(* IEC 61131-3 sources: AXOpen/src/components.rexroth.drives/ctrl/src/AxoIndraDrive (part 2) *)

            _AxisReference ?= AxisRef;

            Messenger.ActivateOnCondition(ULINT#1401,_AxisReference = NULL, eAxoMessageCategory#ProgrammingError);

            IF(_AxisReference = NULL) THEN
                RETURN;
            END_IF;

            Status := FALSE;
            Error	:= FALSE;
            ErrorID :=	DINT#0;
            Valid := FALSE;
            IF Enable OR MC_PowerEnable_PV THEN
                IF _AxisReference^.Data.CheckAccessOK	THEN
                    IF Enable THEN (*	raising edge of ENABLE *)
                        _AxisReference^.Data.PowerOnReq := TRUE;
                    ELSE
                        _AxisReference^.Data.PowerOnReq := FALSE;
                        _AxisReference^.Data.CallNumberCyclic := _AxisReference^.Data.CallNumberCyclic + INT#2;
                    END_IF;
                    _AxisReference^.Data.CallAxis := TRUE;
                    _AxisReference^.Data.ReadOnlyData := FALSE;
                        THIS.FieldBusCommunication(AxisRef := _AxisReference,
                                                    CommandWriteActive=> Dummy);
                    IF _AxisReference^.Data.PowerOK THEN
                        Status	:= TRUE;						(* Status OK*)
                        Valid := TRUE;
                    END_IF;
                    IF _AxisReference^.Data.PowerError = TRUE THEN
                        Error		:= TRUE; 						(*	Set the ERROR-Output *)
                        Valid := TRUE;
                        ErrorID := TO_DINT(_AxisReference^.Data.ErrorID);
                    ELSIF _AxisReference^.Data.CallAxis THEN
                        Error := TRUE;
                        Valid := TRUE;
                        ErrorID := TO_DINT(AXOpen.Components.Rexroth.Drives.eAxoIndraDriveErrorCode#RESOURCE_ERROR);
                    END_IF;
                ELSE
                    Error := TRUE;
                    Valid := TRUE;
                    ErrorID :=TO_DINT( AXOpen.Components.Rexroth.Drives.eAxoIndraDriveErrorCode#RESOURCE_ERROR);
                END_IF;
            END_IF;
            MC_PowerEnable_PV := Enable;
        END_METHOD

        ///<summary>
        /// This method commands the axis to perform the «search home» sequence. The details of this sequence are
        /// manufacturer dependent and can be set by the axis’ parameters. The ‘Position’ input is used to set the absolute
        /// position when reference signal is detected. This method completes at ‘Standstill’ if it was started in ‘Standstill’.
        ///</summary>
        VAR INTERNAL
            MC_HomeExecute_PV					:	BOOL := FALSE;		//Execute - previous value
            MC_HomeCallNumber					: 	INT; 				//Call number of the method MC_Stop
            MC_HomeFirstCall					: 	BOOL;				//First call of the method MC_Stop
            MC_HomeDone_						:	BOOL;
            MC_HomeActive_						:	BOOL;
            MC_HomeCommandAborted_				:	BOOL;
            MC_HomeError_						:	BOOL;
            MC_HomeErrorID_						:	DINT;
            MC_HomeState_						:	UINT;
        END_VAR
        METHOD PUBLIC OVERRIDE MC_Home
            VAR_INPUT
                AxisRef         :   AXOpen.Components.Abstractions.Drives.IAxoAxisReference;
                Execute         :   BOOL;                       //  Start the motion at rising edge
                Position        :   LREAL;                      //  Absolute position when the reference signal is detected
                HommingMode     :   INT;                        //  Required homming mode
                Velocity        :   LREAL;                      //  Value of the maximum ‘Velocity’ (not necessarily reached) [u/s].
                Acceleration    :   LREAL;                      //  Value of the ‘Acceleration’ (always positive) (increasing energy of the motor) [u/s2]
                Deceleration    :   LREAL;                      //  Value of the ‘Deceleration’ (always positive) (decreasing energy of the motor) [u/s2]
            END_VAR
            VAR_OUTPUT
                Done            :   BOOL;                       // Reference known and set sucessfully
                Busy            :   BOOL;                       // The method is not finished and new output values are to be expected
                Active          :   BOOL;                       // Indicates that the method has control on the axis
                CommandAborted  :   BOOL;                       // ‘Command’ is aborted by another command
                Error           :   BOOL;                       // Signals that an error has occurred within the method
                ErrorID         :   DINT;                       // Error identification
             END_VAR
             VAR
                _AxisReference :  REF_TO AXOpen.Components.Rexroth.Drives.AxoIndraDriveAxisReference;

                _ErrorID : DINT;
                _HommingMode: DINT;
                Dummy : BOOL;
                _result : IAxoTaskState;
            END_VAR

            _AxisReference ?= AxisRef;

            Messenger.ActivateOnCondition(ULINT#1402,_AxisReference = NULL, eAxoMessageCategory#ProgrammingError);

            IF(_AxisReference = NULL) THEN
                RETURN;
            END_IF;

            IF Execute AND NOT MC_HomeExecute_PV AND MC_HomeState_ = UINT#0 THEN
                MC_HomeState_ := UINT#10;
            END_IF;
            IF MC_HomeState_ = UINT#10 THEN
                //S-0-0052, Reference distance of encoder 1
                _result := THIS.AxoWriteParameter(ParameterNumber := 52, Value := TO_DINT(Position * EXP(LN(10)* PositionExponent)),ExecutionMode := AXOpen.Components.Abstractions.Drives.eAxoExecutionMode#Immediately, ErrorID =>_ErrorID);
                IF _result.IsDone() THEN
                    MC_HomeState_ := UINT#20;
                END_IF;
                IF _result.HasError() THEN
                    MC_HomeError_ := TRUE;
                    MC_HomeErrorID_ := _ErrorID;
                END_IF;
            END_IF;
            IF MC_HomeState_ = UINT#20 THEN
                AxoWriteParameter_Task.Restore();
                IF(AxoWriteParameter_Task.IsReady()) THEN
                    MC_HomeState_ :=UINT#30;
                    RETURN;
                END_IF;
            END_IF;
            IF MC_HomeState_ = UINT#30 THEN
                IF HommingMode = 0 THEN
                    _HommingMode := 551;
                ELSE
                    _HommingMode := HommingMode;
                END_IF;
                //S-0-0147, Homing parameter
                _result := THIS.AxoWriteParameter(ParameterNumber := 147, Value := _HommingMode ,ExecutionMode := AXOpen.Components.Abstractions.Drives.eAxoExecutionMode#Immediately,ErrorID =>_ErrorID);
                IF _result.IsDone() THEN
                    MC_HomeState_ := UINT#40;
                END_IF;
                IF _result.HasError() THEN
                    MC_HomeError_ := TRUE;
                    MC_HomeErrorID_ := _ErrorID;
                END_IF;
            END_IF;
            IF MC_HomeState_ = UINT#40 THEN
                AxoWriteParameter_Task.Restore();
                IF(AxoWriteParameter_Task.IsReady()) THEN
                    MC_HomeState_ := UINT#50;
                    RETURN;
                END_IF;
            END_IF;
            IF MC_HomeState_ = UINT#50 THEN
                //S-0-0041, Homing velocity
                _result := THIS.AxoWriteParameter(ParameterNumber := 41, Value := TO_DINT(Velocity * EXP(LN(10)*VelocityExponent)) ,ExecutionMode := AXOpen.Components.Abstractions.Drives.eAxoExecutionMode#Immediately, ErrorID =>_ErrorID);
                IF _result.IsDone() THEN
                    MC_HomeState_ :=UINT#60;
                END_IF;
                IF _result.HasError() THEN
                    MC_HomeError_ := TRUE;
                    MC_HomeErrorID_ := _ErrorID;
                END_IF;
            END_IF;
            IF MC_HomeState_ = UINT#60 THEN
                AxoWriteParameter_Task.Restore();
                IF(AxoWriteParameter_Task.IsReady()) THEN
                    MC_HomeState_ :=UINT#70;
                    RETURN;
                END_IF;
            END_IF;
            IF MC_HomeState_ = UINT#70 THEN
                //S-0-0042, Homing acceleration
                _result := THIS.AxoWriteParameter(ParameterNumber := 42, Value := TO_DINT(Acceleration * EXP(LN(10)*AccelerationExponent)) ,ExecutionMode := AXOpen.Components.Abstractions.Drives.eAxoExecutionMode#Immediately, ErrorID =>_ErrorID);
                IF _result.IsDone() THEN
                    MC_HomeState_ := UINT#80;
                END_IF;
                IF _result.HasError() THEN
                    MC_HomeError_ := TRUE;
                    MC_HomeErrorID_ := _ErrorID;
                END_IF;
            END_IF;
            IF MC_HomeState_ = UINT#80 THEN
                AxoWriteParameter_Task.Restore();
                IF(AxoWriteParameter_Task.IsReady()) THEN
                    MC_HomeState_ := UINT#90;
                    RETURN;
                END_IF;
            END_IF;

            IF Execute AND MC_HomeState_ < UINT#90 THEN
                RETURN;
            END_IF;

            (************ start of homing *****************************)
            IF Execute OR MC_HomeExecute_PV  THEN
                MC_HomeFirstCall := TRUE;
                IF _AxisReference^.Data.CheckAccessOK	THEN
                    IF NOT _AxisReference^.Data.PowerOK OR  _AxisReference^.Data.DriveStopReq AND MC_HomeActive_ THEN
                        MC_HomeDone_ := FALSE;
                        MC_HomeActive_ := FALSE;
                        MC_HomeCommandAborted_ := TRUE;
                        _AxisReference^.Data.HomingReq:= FALSE;
                    END_IF;
                    IF Execute AND NOT MC_HomeExecute_PV  THEN
                        IF _AxisReference^.Data.PowerOK AND NOT _AxisReference^.Data.DriveStopReq THEN
                            _AxisReference^.Data.CallNumberCyclic := _AxisReference^.Data.CallNumberCyclic + INT#2;
                            MC_HomeCallNumber := _AxisReference^.Data.CallNumberCyclic;
                            _AxisReference^.Data.WriteCommand:= TRUE;
                            _AxisReference^.Data.HomingReq:= TRUE;
                            _AxisReference^.Data.DriveStopReq:= FALSE;
                            _AxisReference^.Data.DriveHaltReq:= FALSE;
                            _AxisReference^.Data.MoveVelocityReq:= FALSE;
                            _AxisReference^.Data.TorqueControlReq:= FALSE;
                            _AxisReference^.Data.Relative:= FALSE;
                            _AxisReference^.Data.Additive:= FALSE;
                            _AxisReference^.Data.Position := Position;
                            _AxisReference^.Data.Velocity := Velocity;
                            _AxisReference^.Data.Acceleration := Acceleration;
                            _AxisReference^.Data.Deceleration := Deceleration;
                        ELSE
                            MC_HomeError_ := TRUE;
                            MC_HomeErrorID_ := TO_DINT(AXOpen.Components.Rexroth.Drives.eAxoIndraDriveErrorCode#STATE_MACHINE_Error); 	(*State machine MC_HomeError_*)
                        END_IF;
                    END_IF;
                ELSE
                    MC_HomeCallNumber := MC_HomeCallNumber - INT#1;
                    MC_HomeError_ := TRUE;
                    MC_HomeErrorID_ := TO_DINT(AXOpen.Components.Rexroth.Drives.eAxoIndraDriveErrorCode#RESOURCE_Error);
                END_IF;
                IF NOT Execute AND MC_HomeExecute_PV THEN
                    _AxisReference^.Data.HomingReq:= FALSE;
                    MC_HomeCommandAborted_ := FALSE;
                    MC_HomeError_ := FALSE;
                    MC_HomeErrorID_ := TO_DINT(AXOpen.Components.Rexroth.Drives.eAxoIndraDriveErrorCode#NONE_Error);
                END_IF;
            // ELSE
            //     MC_HomeDone_					:= FALSE;
            //     MC_HomeActive_					:= FALSE;
            //     MC_HomeCommandAborted_ 			:= FALSE;
            //     MC_HomeError_					:= FALSE;
            //     MC_HomeErrorID_ 				:= AXOpen.Components.Rexroth.Drives.eAxoIndraDriveErrorCode#NONE_Error;
            //     MC_HomeState_ 					:= UINT#0;
            END_IF;
            (*************** detection of command finished *******************)
            IF MC_HomeFirstCall THEN
                IF MC_HomeCallNumber = _AxisReference^.Data.CallNumberCyclic THEN
                    _AxisReference^.Data.CallAxis := TRUE;
                    _AxisReference^.Data.ReadOnlyData := FALSE;
                    THIS.FieldBusCommunication(	AxisRef := _AxisReference,CommandWriteActive=> Dummy);
                    IF NOT _AxisReference^.Data.CommandWriteActive THEN
                         IF _AxisReference^.Data.SetpointReached THEN
                            MC_HomeDone_ := TRUE;
                            MC_HomeActive_ := FALSE;
                            _AxisReference^.Data.HomingReq:= FALSE;
                        ELSE
                            MC_HomeActive_ := TRUE;
                        END_IF;
                        IF _AxisReference^.Data.Error THEN
                            MC_HomeDone_ 	:= FALSE;
                            MC_HomeActive_ 	:= FALSE;
                            MC_HomeError_ 	:= TRUE;
                            MC_HomeErrorID_ := TO_DINT(_AxisReference^.Data.ErrorID);
                        ELSIF _AxisReference^.Data.CallAxis THEN
                            MC_HomeError_ := TRUE;
                            MC_HomeErrorID_ := TO_DINT(AXOpen.Components.Rexroth.Drives.eAxoIndraDriveErrorCode#RESOURCE_ERROR);
                        END_IF;
                    END_IF;
                END_IF;
                (************** reset of outputs *************************************)
                IF Execute = FALSE THEN
                    _AxisReference^.Data.HomingReq:= FALSE;
                    (****** reset outputs ***********)
                    MC_HomeDone_ := FALSE;
                    MC_HomeActive_ := FALSE;
                    MC_HomeCommandAborted_ := FALSE;
                    MC_HomeError_ := FALSE;
                    MC_HomeErrorID_ :=	TO_DINT(AXOpen.Components.Rexroth.Drives.eAxoIndraDriveErrorCode#NONE_ERROR);
                    MC_HomeState_ := UINT#0;
                    IF MC_HomeCallNumber = _AxisReference^.Data.CallNumberCyclic THEN
                        _AxisReference^.Data.CallAxis := TRUE;
                        _AxisReference^.Data.ReadOnlyData := FALSE;
                        THIS.FieldBusCommunication(	AxisRef := _AxisReference,CommandWriteActive=> Dummy);
                        IF _AxisReference^.Data.SetpointReached THEN
                            MC_HomeDone_ := TRUE;
                            MC_HomeCallNumber := MC_HomeCallNumber - INT#1; (*Reset MC_HomeCallNumber because reset MC_HomeDone_ *)
                        END_IF;
                    END_IF;
                END_IF;
            END_IF;

            MC_HomeExecute_PV 	:=	Execute;
            Done				:=	MC_HomeDone_;
            Active 				:=	MC_HomeActive_;
            CommandAborted 		:=	MC_HomeCommandAborted_;
            Error 				:=	MC_HomeError_;
            ErrorID 			:=	MC_HomeErrorID_;
            Busy				:=	MC_HomeActive_ AND NOT Done AND NOT Error;

        END_METHOD

        ///<summary>
        /// This method commands a controlled motion stop and transfers the axis to the state ‘Stopping’. It aborts any
        /// ongoing method execution. While the axis is in state ‘Stopping’, no other method can perform any motion on the
        /// same axis.
        ///</summary>
        VAR INTERNAL
            MC_StopExecute_PV					: 	BOOL;				//Execute - previous value
            MC_StopCallNumber					:	INT;				//Call number of the method MC_Stop
            MC_StopFirstCall					: 	BOOL;				//First call of the method MC_Stop
        END_VAR
        METHOD PUBLIC OVERRIDE MC_Stop
            VAR_INPUT
                AxisRef         :   AXOpen.Components.Abstractions.Drives.IAxoAxisReference;
                Execute         :   BOOL;                       //  Start the action at rising edge
                Deceleration    :   LREAL;                      //  Value of the ‘Deceleration’ [u/s2]
                Jerk            :   LREAL;                      //  Value of the ‘Jerk’ [u/s3]
            END_VAR
            VAR_OUTPUT
                Done            :   BOOL;                       // Zero velocity reached
                Busy            :   BOOL;                       // The method is not finished and new output values are to be expected
                Active          :   BOOL;                       // Indicates that the method has control on the axis
                CommandAborted  :   BOOL;                       // ‘Command’ is aborted by switching off power (only possibility to abort)
                Error           :   BOOL;                       // Signals that an error has occurred within the method
                ErrorID         :   DINT;                       // Error identification
             END_VAR
             VAR
                _AxisReference :  REF_TO AXOpen.Components.Rexroth.Drives.AxoIndraDriveAxisReference;
                Dummy : BOOL;
            END_VAR

            _AxisReference ?= AxisRef;

            Messenger.ActivateOnCondition(ULINT#1403,_AxisReference = NULL, eAxoMessageCategory#ProgrammingError);

            IF(_AxisReference = NULL) THEN
                RETURN;
            END_IF;

            Done := FALSE;
            IF Execute OR MC_StopExecute_PV THEN 								(* Execute = Stop to Drive *)
                IF Execute THEN
                    MC_StopFirstCall := TRUE;
                    IF _AxisReference^.Data.CheckAccessOK THEN
                        IF Execute AND NOT MC_StopExecute_PV THEN
                            _AxisReference^.Data.CallNumberCyclic := _AxisReference^.Data.CallNumberCyclic + INT#2;
                            MC_StopCallNumber := _AxisReference^.Data.CallNumberCyclic;
                        END_IF;
                        Active := TRUE;
                        _AxisReference^.Data.DriveStopReq := TRUE;
                        _AxisReference^.Data.Deceleration := Deceleration;
                        _AxisReference^.Data.Jerk := Jerk;
                        _AxisReference^.Data.CallAxis := TRUE;
                        _AxisReference^.Data.ReadOnlyData := FALSE;
                        _AxisReference^.Data.HomingReq:= FALSE;
                        THIS.FieldBusCommunication(AxisRef := _AxisReference,
                                                CommandWriteActive=> Dummy);
                        IF 	_AxisReference^.Data.StopError AND MC_StopCallNumber = _AxisReference^.Data.CallNumberCyclic THEN
                            Error		:= TRUE; 						(*	Set the ERROR-Output *)
                            ErrorID :=	TO_DINT(_AxisReference^.Data.ErrorID);
                        ELSIF _AxisReference^.Data.CallAxis THEN
                            Active := FALSE;
                            Error := TRUE;
                            ErrorID := TO_DINT(AXOpen.Components.Rexroth.Drives.eAxoIndraDriveErrorCode#RESOURCE_ERROR);
                        END_IF;
                    ELSE
                        MC_StopCallNumber := MC_StopCallNumber - INT#1;
                        Error := TRUE;
                        ErrorID := TO_DINT(AXOpen.Components.Rexroth.Drives.eAxoIndraDriveErrorCode#RESOURCE_ERROR);
                    END_IF;
                END_IF;
                IF _AxisReference^.Data.Stopped THEN
                    Done := TRUE;
                    Active := FALSE;
                END_IF;
                IF NOT Execute AND MC_StopExecute_PV THEN
                    _AxisReference^.Data.DriveStopReq := FALSE;
                END_IF;
            ELSE
                Error	:= FALSE;
                ErrorID :=	DINT#0;
            END_IF;
            IF NOT Execute AND MC_StopFirstCall AND Active THEN
                IF MC_StopCallNumber = _AxisReference^.Data.CallNumberCyclic THEN
                    _AxisReference^.Data.CallAxis := TRUE;
                    _AxisReference^.Data.ReadOnlyData := FALSE;
                        THIS.FieldBusCommunication(AxisRef:= _AxisReference,
                                                CommandWriteActive=> Dummy);
                    IF _AxisReference^.Data.Stopped THEN
                        Done := TRUE;
                        Active := FALSE;
                        MC_StopCallNumber := MC_StopCallNumber -INT#1;
                    END_IF;
                ELSE
                    Done := FALSE;
                    Active := FALSE;
                    CommandAborted := TRUE;
                END_IF;
            ELSE
                CommandAborted := FALSE;
            END_IF;
            MC_StopExecute_PV := Execute;
            Busy := Execute AND NOT Done AND NOT Error;

            ;
        END_METHOD

        ///<summary>
        /// This method commands a controlled motion stop. The axis is moved to the state ‘DiscreteMotion’, until the
        /// velocity is zero. With the ‘Done’ output set, the state is transferred to ‘Standstill’.
        ///</summary>
        VAR INTERNAL
            MC_HaltExecute_PV					: 	BOOL;				//Execute - previous value
            MC_HaltCallNumber					:	INT;				//Call number of the method MC_Halt
            MC_HaltFirstCall					: 	BOOL;				//First call of the method MC_Halt
            MC_HaltDone_						:	BOOL;
            MC_HaltActive_						:	BOOL;
            MC_HaltCommandAborted_				:	BOOL;
            MC_HaltError_						:	BOOL;
            MC_HaltErrorID_						:	eAxoIndraDriveErrorCode;
        END_VAR
        METHOD PUBLIC OVERRIDE MC_Halt
            VAR_INPUT
                AxisRef         :   AXOpen.Components.Abstractions.Drives.IAxoAxisReference;
                Execute         :   BOOL;                       //  Start the action at rising edge
                Deceleration    :   LREAL;                      //  Value of the ‘Deceleration’ [u/s2]
                Jerk            :   LREAL;                      //  Value of the ‘Jerk’ [u/s3]
            END_VAR
            VAR_OUTPUT
                Done            :   BOOL;                       // Zero velocity reached
                Busy            :   BOOL;                       // The method is not finished and new output values are to be expected
                Active          :   BOOL;                       // Indicates that the method has control on the axis
                CommandAborted  :   BOOL;                       // ‘Command’ is aborted by switching off power (only possibility to abort)
                Error           :   BOOL;                       // Signals that an error has occurred within the method
                ErrorID         :   DINT;                       // Error identification
            END_VAR
            VAR
                _AxisReference :  REF_TO AXOpen.Components.Rexroth.Drives.AxoIndraDriveAxisReference;
                Dummy : BOOL;
            END_VAR

            _AxisReference ?= AxisRef;

            Messenger.ActivateOnCondition(ULINT#1404,_AxisReference = NULL, eAxoMessageCategory#ProgrammingError);

            IF(_AxisReference = NULL) THEN
                RETURN;
            END_IF;
            IF Execute OR MC_HaltExecute_PV THEN 								(* Execute = Halt to Drive *)
                MC_HaltFirstCall := TRUE;
                IF _AxisReference^.Data.CheckAccessOK THEN
                    IF NOT MC_HaltDone_ THEN
                        IF Execute AND NOT MC_HaltExecute_PV THEN
                            MC_HaltDone_ := FALSE;
                            _AxisReference^.Data.CallNumberCyclic := _AxisReference^.Data.CallNumberCyclic + INT#2;
                            MC_HaltCallNumber := _AxisReference^.Data.CallNumberCyclic;
                            _AxisReference^.Data.DriveHaltReq := TRUE;
                            _AxisReference^.Data.HomingReq:= FALSE;
                            _AxisReference^.Data.MoveVelocityReq:= FALSE;
                            _AxisReference^.Data.TorqueControlReq:= FALSE;
                            _AxisReference^.Data.Relative:= FALSE;
                            _AxisReference^.Data.Additive:= FALSE;
                            _AxisReference^.Data.Deceleration := Deceleration;
                            _AxisReference^.Data.Jerk := Jerk;
                        END_IF;
                        MC_HaltActive_ := TRUE;
                        _AxisReference^.Data.CallAxis := TRUE;
                        _AxisReference^.Data.ReadOnlyData := FALSE;
                        _AxisReference^.Data.HomingReq:= FALSE;
                        THIS.FieldBusCommunication(AxisRef:= _AxisReference,
                                                CommandWriteActive=> Dummy);
                        IF 	_AxisReference^.Data.StopError AND MC_HaltCallNumber = _AxisReference^.Data.CallNumberCyclic THEN
                            MC_HaltError_		:= TRUE; 						(*	Set the ERROR-Output *)
                            MC_HaltErrorID_ :=	_AxisReference^.Data.ErrorID;
                        ELSIF _AxisReference^.Data.CallAxis THEN
                            MC_HaltActive_ := FALSE;
                            MC_HaltError_ := TRUE;
                            MC_HaltErrorID_ := AXOpen.Components.Rexroth.Drives.eAxoIndraDriveErrorCode#RESOURCE_ERROR;
                        END_IF;
                    END_IF;
                ELSE
                    MC_HaltCallNumber := MC_HaltCallNumber - INT#1;
                    MC_HaltError_ := TRUE;
                    MC_HaltErrorID_ := AXOpen.Components.Rexroth.Drives.eAxoIndraDriveErrorCode#RESOURCE_ERROR;
                END_IF;
                IF _AxisReference^.Fieldbus_In.InStandstill THEN
                    MC_HaltDone_ := TRUE;
                    MC_HaltActive_ := FALSE;
                    _AxisReference^.Data.DriveHaltReq := FALSE;
                END_IF;
                IF NOT Execute AND MC_HaltExecute_PV THEN
                    _AxisReference^.Data.DriveHaltReq := FALSE;
                END_IF;
            ELSE
                MC_HaltDone_ := FALSE;
                MC_HaltActive_ := FALSE;
                MC_HaltError_		:= FALSE;
                MC_HaltErrorID_ :=	AXOpen.Components.Rexroth.Drives.eAxoIndraDriveErrorCode#NONE_ERROR;
            END_IF;
            IF NOT Execute AND MC_HaltFirstCall AND MC_HaltActive_ THEN
                IF MC_HaltCallNumber = _AxisReference^.Data.CallNumberCyclic THEN
                    _AxisReference^.Data.CallAxis := TRUE;
                    _AxisReference^.Data.ReadOnlyData := FALSE;
                                    THIS.FieldBusCommunication(AxisRef:= _AxisReference,
                                                CommandWriteActive=> Dummy);
                    IF _AxisReference^.Data.Stopped THEN
                        MC_HaltDone_ := TRUE;
                        MC_HaltActive_ := FALSE;
                        MC_HaltCallNumber := MC_HaltCallNumber - INT#1;
                    END_IF;
                ELSE
                    MC_HaltDone_ := FALSE;
                    MC_HaltActive_ := FALSE;
                    MC_HaltCommandAborted_ := TRUE;
                END_IF;
            ELSE
                MC_HaltCommandAborted_ := FALSE;
            END_IF;
            MC_HaltExecute_PV := Execute;

            Done			:=  MC_HaltDone_;
            Busy := Execute AND NOT Done AND NOT Error;
            Active			:=  MC_HaltActive_;
            CommandAborted	:=  MC_HaltCommandAborted_;
            Error			:=  MC_HaltError_;
            ErrorID			:=  TO_DINT(MC_HaltErrorID_);

        END_METHOD

        ///<summary>
        /// This method commands a controlled motion to a specified absolute position.
        ///<summary>
        VAR INTERNAL
            MC_MoveAbsoluteExecute_PV			: 	BOOL := FALSE;		//Execute - previous value
            MC_MoveAbsoluteDone_PV				:	BOOL := FALSE;		//Done - previous value
            MC_MoveAbsoluteCallNumber			: 	INT; 				//Call number of the method MC_MoveAbsolute
            MC_MoveAbsoluteFirstCall			: 	BOOL;				//First call of the method MC_MoveAbsolute
            MC_MoveAbsoluteDone_				:	BOOL;
            MC_MoveAbsoluteActive_				:	BOOL;
            MC_MoveAbsoluteCommandAborted_		:	BOOL;
            MC_MoveAbsoluteError_				:   BOOL;
            MC_MoveAbsoluteErrorID_				:   eAxoIndraDriveErrorCode;
            MC_MoveAbsoluteContinuousUpdate_PV  :   BOOL;
        END_VAR
        METHOD PUBLIC OVERRIDE MC_MoveAbsolute
            VAR_INPUT
                AxisRef         :   AXOpen.Components.Abstractions.Drives.IAxoAxisReference;
                Execute         :   BOOL;                       //  Start the motion at rising edge
                ContinuousUpdate:   BOOL;                       //  Activate ‘ContinuousUpdate’ - target parameters should be changed during movement
                Position        :   LREAL;                      //  Commanded ‘Position’ for the motion (in technical unit [u]) (negative or positive)
                Velocity        :   LREAL;                      //  Value of the maximum ‘Velocity’ (not necessarily reached) [u/s].
                Acceleration    :   LREAL;                      //  Value of the ‘Acceleration’ (always positive) (increasing energy of the motor) [u/s2]
                Deceleration    :   LREAL;                      //  Value of the ‘Deceleration’ (always positive) (decreasing energy of the motor) [u/s2]
                Jerk            :   LREAL;                      //  Value of the ‘Jerk’ [u/s3]
                Direction       :   AXOpen.Components.Abstractions.Drives.eAxoDriveDirection;         //  Enum type (1-of-4 values: PositiveDirection, ShortestWay, NegativeDirection, CurrentDirection)
            END_VAR
            VAR_OUTPUT
                Done            :   BOOL;                       // Commanded position finally reached
                Busy            :   BOOL;                       // The method is not finished and new output values are to be expected
                Active          :   BOOL;                       // Indicates that the method has control on the axis
                CommandAborted  :   BOOL;                       // ‘Command’ is aborted by another command
                Error           :   BOOL;                       // Signals that an error has occurred within the method
                ErrorID         :   DINT;                       // Error identification
            END_VAR
            VAR
                _AxisReference :  REF_TO AXOpen.Components.Rexroth.Drives.AxoIndraDriveAxisReference;
                Dummy : BOOL;
            END_VAR

            _AxisReference ?= AxisRef;

            Messenger.ActivateOnCondition(ULINT#1405,_AxisReference = NULL, eAxoMessageCategory#ProgrammingError);

            IF(_AxisReference = NULL) THEN
                RETURN;
            END_IF;

            IF Execute OR (NOT Execute AND MC_MoveAbsoluteExecute_PV) THEN (*detection of falling edge execute*)
                MC_MoveAbsoluteFirstCall := TRUE;
                IF _AxisReference^.Data.CheckAccessOK	THEN
                    IF Execute AND NOT MC_MoveAbsoluteExecute_PV THEN (*	raising edge of EXECUTE *)
                        MC_MoveAbsoluteContinuousUpdate_PV := ContinuousUpdate;
                        _AxisReference^.Data.CallNumberCyclic := _AxisReference^.Data.CallNumberCyclic + INT#2;
                        MC_MoveAbsoluteCallNumber := _AxisReference^.Data.CallNumberCyclic;
                        _AxisReference^.Data.WriteCommand:= TRUE;
                        _AxisReference^.Data.HomingReq:= FALSE;
            (*			Axis.Data.DriveStopReq:= FALSE;*)
                        _AxisReference^.Data.DriveHaltReq := FALSE;
                        _AxisReference^.Data.MoveVelocityReq:= FALSE;
                        _AxisReference^.Data.TorqueControlReq:= FALSE;
                        _AxisReference^.Data.Relative:= FALSE;
                        _AxisReference^.Data.Additive:= FALSE;
                        _AxisReference^.Data.Position := Position;
                        _AxisReference^.Data.Velocity := Velocity;
                        _AxisReference^.Data.Acceleration := Acceleration;
                        _AxisReference^.Data.Deceleration := Deceleration;
                        _AxisReference^.Data.Jerk:= Jerk;
                        MC_MoveAbsoluteDone_ := FALSE;
                        MC_MoveAbsoluteActive_ := TRUE;
                        MC_MoveAbsoluteError_ := FALSE;
                        MC_MoveAbsoluteErrorID_ :=	AXOpen.Components.Rexroth.Drives.eAxoIndraDriveErrorCode#NONE_ERROR;
                    END_IF;
                ELSE
                    MC_MoveAbsoluteCallNumber := MC_MoveAbsoluteCallNumber - INT#1;
                    MC_MoveAbsoluteError_ := TRUE;
                    MC_MoveAbsoluteErrorID_ := AXOpen.Components.Rexroth.Drives.eAxoIndraDriveErrorCode#RESOURCE_ERROR;
                END_IF;
            END_IF;
            (************** reset of outputs *************************************)
            IF Execute = FALSE THEN
                MC_MoveAbsoluteCommandAborted_ := FALSE;
                MC_MoveAbsoluteDone_ := FALSE;
                MC_MoveAbsoluteError_ := FALSE;
                MC_MoveAbsoluteErrorID_ :=	AXOpen.Components.Rexroth.Drives.eAxoIndraDriveErrorCode#NONE_ERROR;
            END_IF;
            (*************** detection of command finished *******************)
            IF MC_MoveAbsoluteFirstCall THEN
                IF MC_MoveAbsoluteCallNumber = _AxisReference^.Data.CallNumberCyclic THEN
                    MC_MoveAbsoluteActive_ := TRUE;
                    _AxisReference^.Data.CallAxis := TRUE;
                    _AxisReference^.Data.ReadOnlyData := FALSE;
                    THIS.FieldBusCommunication(AxisRef := _AxisReference,CommandWriteActive=> Dummy);
                    IF NOT _AxisReference^.Data.CommandWriteActive THEN
                        MC_MoveAbsoluteActive_ := TRUE;
                        IF MC_MoveAbsoluteContinuousUpdate_PV AND
                            (_AxisReference^.Data.Position <> Position OR
                            _AxisReference^.Data.Velocity <> Velocity OR
                            _AxisReference^.Data.Acceleration <> Acceleration OR
                            _AxisReference^.Data.Deceleration <> Deceleration OR
                            _AxisReference^.Data.Jerk <> Jerk ) THEN
                            _AxisReference^.Data.Position := Position;
                            _AxisReference^.Data.Velocity := Velocity;
                            _AxisReference^.Data.Acceleration := Acceleration;
                            _AxisReference^.Data.Deceleration := Deceleration;
                            _AxisReference^.Data.Jerk:= Jerk;
                            _AxisReference^.Data.WriteCommand := TRUE;
                            _AxisReference^.Data.CallAxis := TRUE;
                            _AxisReference^.Data.ReadOnlyData := FALSE;
                            THIS.FieldBusCommunication(AxisRef := _AxisReference,CommandWriteActive=> Dummy);
                            RETURN;
                        END_IF;

                        IF _AxisReference^.Data.SetpointReached THEN
                            MC_MoveAbsoluteDone_ := TRUE;
                            MC_MoveAbsoluteActive_ := FALSE;
                            MC_MoveAbsoluteCallNumber := MC_MoveAbsoluteCallNumber - INT#1; (*Reset MC_MoveAbsoluteCallNumber because reset Done *)
                        END_IF;
                    END_IF;
                    IF _AxisReference^.Data.Error THEN
                        MC_MoveAbsoluteCallNumber := MC_MoveAbsoluteCallNumber - INT#1;
                        MC_MoveAbsoluteActive_ := FALSE;
                        MC_MoveAbsoluteError_ := TRUE;
                        MC_MoveAbsoluteErrorID_ := _AxisReference^.Data.ErrorID;
                    ELSIF _AxisReference^.Data.CallAxis THEN
                        MC_MoveAbsoluteCallNumber := MC_MoveAbsoluteCallNumber - INT#1;
                        MC_MoveAbsoluteActive_ := FALSE;
                        MC_MoveAbsoluteError_ := TRUE;
                        MC_MoveAbsoluteErrorID_ := AXOpen.Components.Rexroth.Drives.eAxoIndraDriveErrorCode#RESOURCE_ERROR;
                    END_IF;
                ELSE
                    (*************** detection of command aborted ********************)
                    IF MC_MoveAbsoluteActive_ THEN
                        MC_MoveAbsoluteCommandAborted_ := TRUE;
                    END_IF;
                    MC_MoveAbsoluteActive_ := FALSE;
                END_IF;
            END_IF;

            IF NOT ContinuousUpdate THEN
                MC_MoveAbsoluteContinuousUpdate_PV := FALSE;
            END_IF;
            MC_MoveAbsoluteExecute_PV := Execute;

            Done			:=	MC_MoveAbsoluteDone_;
            Busy			:=	Execute AND NOT Done AND NOT Error;
            Active			:=	MC_MoveAbsoluteActive_;
            CommandAborted	:=	MC_MoveAbsoluteCommandAborted_;
            Error			:=	MC_MoveAbsoluteError_;
            ErrorID			:=	TO_DINT(MC_MoveAbsoluteErrorID_);

        END_METHOD

        ///<summary>
        /// This method  commands a controlled motion of a specified distance relative to the set position at the time of the execution.
        ///<summary>
        VAR INTERNAL
            MC_MoveRelativeExecute_PV			: 	BOOL := FALSE;		//Execute - previous value
            MC_MoveRelativeDone_PV				:	BOOL := FALSE;		//Done - previous value
            MC_MoveRelativeCallNumber			: 	INT; 				//Call number of the method MC_MoveRelative
            MC_MoveRelativeFirstCall			: 	BOOL;				//First call of the method MC_MoveRelative
            MC_MoveRelativeDone_				:	BOOL;
            MC_MoveRelativeActive_				:	BOOL;
            MC_MoveRelativeCommandAborted_		:	BOOL;
            MC_MoveRelativeError_				:   BOOL;
            MC_MoveRelativeErrorID_				:   eAxoIndraDriveErrorCode;
            MC_MoveRelativeContinuousUpdate_PV  :   BOOL;
            MC_MoveRelativeDistance_PV          :   LREAL;
        END_VAR
        METHOD PUBLIC OVERRIDE MC_MoveRelative
            VAR_INPUT
                AxisRef         :   AXOpen.Components.Abstractions.Drives.IAxoAxisReference;
                Execute         :   BOOL;                       //  Start the motion at rising edge
                ContinuousUpdate:   BOOL;                       //  Activate ‘ContinuousUpdate’ - target parameters should be changed during movement
                Distance        :   LREAL;                      //  Relative distance for the motion (in technical unit [u]
                Velocity        :   LREAL;                      //  Value of the maximum ‘Velocity’ (not necessarily reached) [u/s].
                Acceleration    :   LREAL;                      //  Value of the ‘Acceleration’ (always positive) (increasing energy of the motor) [u/s2]
                Deceleration    :   LREAL;                      //  Value of the ‘Deceleration’ (always positive) (decreasing energy of the motor) [u/s2]
                Jerk            :   LREAL;                      //  Value of the ‘Jerk’ [u/s3]
            END_VAR
            VAR_OUTPUT
                Done            :   BOOL;                       // Commanded distance reached
                Busy            :   BOOL;                       // The method is not finished and new output values are to be expected
                Active          :   BOOL;                       // Indicates that the method has control on the axis
                CommandAborted  :   BOOL;                       // ‘Command’ is aborted by another command
                Error           :   BOOL;                       // Signals that an error has occurred within the method
                ErrorID         :   DINT;                       // Error identification
            END_VAR
            VAR
                _AxisReference :  REF_TO AXOpen.Components.Rexroth.Drives.AxoIndraDriveAxisReference;
                Dummy : BOOL;
            END_VAR

            _AxisReference ?= AxisRef;

            Messenger.ActivateOnCondition(ULINT#1406,_AxisReference = NULL, eAxoMessageCategory#ProgrammingError);

            IF(_AxisReference = NULL) THEN
                RETURN;
            END_IF;

            IF Execute OR (NOT Execute AND MC_MoveRelativeExecute_PV) THEN (*detection of falling edge execute*)
                MC_MoveRelativeFirstCall := TRUE;
                IF _AxisReference^.Data.CheckAccessOK	THEN
                    IF Execute AND NOT MC_MoveRelativeExecute_PV THEN (*	raising edge of EXECUTE *)
                        MC_MoveRelativeDistance_PV := Distance;
                        MC_MoveRelativeContinuousUpdate_PV := ContinuousUpdate;
                        _AxisReference^.Data.CallNumberCyclic := _AxisReference^.Data.CallNumberCyclic + INT#2;
                        MC_MoveRelativeCallNumber := _AxisReference^.Data.CallNumberCyclic;
                        _AxisReference^.Data.WriteCommand:= TRUE;
                        _AxisReference^.Data.HomingReq:= FALSE;
            (*			Axis.Data.DriveStopReq:= FALSE;*)
                        _AxisReference^.Data.DriveHaltReq := FALSE;
                        _AxisReference^.Data.MoveVelocityReq:= FALSE;
                        _AxisReference^.Data.TorqueControlReq:= FALSE;
                        _AxisReference^.Data.Relative:= TRUE;
                        _AxisReference^.Data.Additive:= TRUE;
                        _AxisReference^.Data.Position := Distance;
                        _AxisReference^.Data.Velocity := Velocity;
                        _AxisReference^.Data.Acceleration := Acceleration;
                        _AxisReference^.Data.Deceleration := Deceleration;
                        _AxisReference^.Data.Jerk:= Jerk;
                        MC_MoveRelativeDone_ := FALSE;
                        MC_MoveRelativeActive_ := TRUE;
                        MC_MoveRelativeError_ := FALSE;
                        MC_MoveRelativeErrorID_ :=	AXOpen.Components.Rexroth.Drives.eAxoIndraDriveErrorCode#NONE_ERROR;
                    END_IF;
                ELSE
                    MC_MoveRelativeCallNumber := MC_MoveRelativeCallNumber - INT#1;
                    MC_MoveRelativeError_ := TRUE;
                    MC_MoveRelativeErrorID_ := AXOpen.Components.Rexroth.Drives.eAxoIndraDriveErrorCode#RESOURCE_ERROR;
                END_IF;
            END_IF;
            (************** reset of outputs *************************************)
            IF Execute = FALSE THEN
                MC_MoveRelativeCommandAborted_ := FALSE;
                MC_MoveRelativeDone_ := FALSE;
                MC_MoveRelativeError_ := FALSE;
                MC_MoveRelativeErrorID_ :=	AXOpen.Components.Rexroth.Drives.eAxoIndraDriveErrorCode#NONE_ERROR;
                MC_MoveRelativeDistance_PV := 0;
            END_IF;
            (*************** detection of command finished *******************)
            IF MC_MoveRelativeFirstCall THEN
                IF MC_MoveRelativeCallNumber = _AxisReference^.Data.CallNumberCyclic THEN
                    MC_MoveRelativeActive_ := TRUE;
                    _AxisReference^.Data.CallAxis := TRUE;
                    _AxisReference^.Data.ReadOnlyData := FALSE;
                    THIS.FieldBusCommunication(AxisRef := _AxisReference,CommandWriteActive=> Dummy);
                    IF NOT _AxisReference^.Data.CommandWriteActive THEN
                        MC_MoveRelativeActive_ := TRUE;
                        IF MC_MoveRelativeContinuousUpdate_PV AND
                            (MC_MoveRelativeDistance_PV<> Distance OR
                            _AxisReference^.Data.Velocity <> Velocity OR
                            _AxisReference^.Data.Acceleration <> Acceleration OR
                            _AxisReference^.Data.Deceleration <> Deceleration OR
                            _AxisReference^.Data.Jerk <> Jerk ) THEN
                            _AxisReference^.Data.Position := Distance-MC_MoveRelativeDistance_PV;
                            _AxisReference^.Data.Velocity := Velocity;
                            _AxisReference^.Data.Acceleration := Acceleration;
                            _AxisReference^.Data.Deceleration := Deceleration;
                            _AxisReference^.Data.Jerk:= Jerk;
                            _AxisReference^.Data.WriteCommand := TRUE;
                            _AxisReference^.Data.CallAxis := TRUE;
                            _AxisReference^.Data.ReadOnlyData := FALSE;
                            MC_MoveRelativeDistance_PV := Distance;
                            THIS.FieldBusCommunication(AxisRef := _AxisReference,CommandWriteActive=> Dummy);
                            RETURN;
                        END_IF;

                        IF _AxisReference^.Data.SetpointReached THEN
                            MC_MoveRelativeDone_ := TRUE;
                            MC_MoveRelativeActive_ := FALSE;
                            MC_MoveRelativeCallNumber := MC_MoveRelativeCallNumber - INT#1; (*Reset MC_MoveRelativeCallNumber because reset Done *)
                        END_IF;
                    END_IF;
                    IF _AxisReference^.Data.Error THEN
                        MC_MoveRelativeCallNumber := MC_MoveRelativeCallNumber - INT#1;
                        MC_MoveRelativeActive_ := FALSE;
                        MC_MoveRelativeError_ := TRUE;
                        MC_MoveRelativeErrorID_ := _AxisReference^.Data.ErrorID;
                    ELSIF _AxisReference^.Data.CallAxis THEN
                        MC_MoveRelativeCallNumber := MC_MoveRelativeCallNumber - INT#1;
                        MC_MoveRelativeActive_ := FALSE;
                        MC_MoveRelativeError_ := TRUE;
                        MC_MoveRelativeErrorID_ := AXOpen.Components.Rexroth.Drives.eAxoIndraDriveErrorCode#RESOURCE_ERROR;
                    END_IF;
                ELSE
                    (*************** detection of command aborted ********************)
                    IF MC_MoveRelativeActive_ THEN
                        MC_MoveRelativeCommandAborted_ := TRUE;
                    END_IF;
                    MC_MoveRelativeActive_ := FALSE;
                END_IF;
            END_IF;

            IF NOT ContinuousUpdate THEN
                MC_MoveRelativeContinuousUpdate_PV := FALSE;
            END_IF;
            MC_MoveRelativeExecute_PV := Execute;

            Done			:=	MC_MoveRelativeDone_;
            Busy			:=	Execute AND NOT Done AND NOT Error;
            Active			:=	MC_MoveRelativeActive_;
            CommandAborted	:=	MC_MoveRelativeCommandAborted_;
            Error			:=	MC_MoveRelativeError_;
            ErrorID			:=	TO_DINT(MC_MoveRelativeErrorID_);
        END_METHOD

        ///<summary>
        /// This method commands a controlled motion of a specified relative distance additional to the most recent
        /// commanded position in the axis state ‘DiscreteMotion’. The most recent commanded position may be the result of a
        /// previous MC_MoveAdditive motion which was aborted. If the method is activated in the axis state ‘ContinuousMotion’, the
        /// specified relative distance is added to the set position at the time of the execution.
        ///<summary>
        VAR INTERNAL
            MC_MoveAdditiveExecute_PV			: 	BOOL := FALSE;		//Execute - previous value
            MC_MoveAdditiveDone_PV				:	BOOL := FALSE;		//Done - previous value
            MC_MoveAdditiveCallNumber			: 	INT; 				//Call number of the method MC_MoveAdditive
            MC_MoveAdditiveFirstCall			: 	BOOL;				//First call of the method MC_MoveAdditive
            MC_MoveAdditiveDone_				:	BOOL;
            MC_MoveAdditiveActive_				:	BOOL;
            MC_MoveAdditiveCommandAborted_		:	BOOL;
            MC_MoveAdditiveError_				:	BOOL;
            MC_MoveAdditiveErrorID_				:	eAxoIndraDriveErrorCode;
            MC_MoveAdditiveContinuousUpdate_PV  :   BOOL;
            MC_MoveAdditiveDistance_PV          :   LREAL;
        END_VAR
        METHOD PUBLIC OVERRIDE MC_MoveAdditive
            VAR_INPUT
                AxisRef         :   AXOpen.Components.Abstractions.Drives.IAxoAxisReference;
                Execute         :   BOOL;                       //  Start the motion at rising edge
                ContinuousUpdate:   BOOL;                       //  Activate ‘ContinuousUpdate’ - target parameters should be changed during movement
                Distance        :   LREAL;                      //  Relative distance for the motion (in technical unit [u]
                Velocity        :   LREAL;                      //  Value of the maximum ‘Velocity’ (not necessarily reached) [u/s].
                Acceleration    :   LREAL;                      //  Value of the ‘Acceleration’ (always positive) (increasing energy of the motor) [u/s2]
                Deceleration    :   LREAL;                      //  Value of the ‘Deceleration’ (always positive) (decreasing energy of the motor) [u/s2]
                Jerk            :   LREAL;                      //  Value of the ‘Jerk’ [u/s3]
            END_VAR
            VAR_OUTPUT
                Done            :   BOOL;                       // Commanded distance reached
                Busy            :   BOOL;                       // The method is not finished and new output values are to be expected
                Active          :   BOOL;                       // Indicates that the method has control on the axis
                CommandAborted  :   BOOL;                       // ‘Command’ is aborted by another command
                Error           :   BOOL;                       // Signals that an error has occurred within the method
                ErrorID         :   DINT;                       // Error identification
            END_VAR
            VAR
                _AxisReference :  REF_TO AXOpen.Components.Rexroth.Drives.AxoIndraDriveAxisReference;
                Dummy : BOOL;
            END_VAR

            _AxisReference ?= AxisRef;

            Messenger.ActivateOnCondition(ULINT#1407,_AxisReference = NULL, eAxoMessageCategory#ProgrammingError);

            IF(_AxisReference = NULL) THEN
                RETURN;
            END_IF;

            IF Execute OR (NOT Execute AND MC_MoveAdditiveExecute_PV) THEN (*detection of falling edge execute*)
                MC_MoveAdditiveFirstCall := TRUE;
                IF _AxisReference^.Data.CheckAccessOK	THEN
                    IF Execute AND NOT MC_MoveAdditiveExecute_PV THEN (*	raising edge of EXECUTE *)
                        MC_MoveAdditiveDistance_PV := Distance;
                        MC_MoveAdditiveContinuousUpdate_PV := ContinuousUpdate;
                        _AxisReference^.Data.CallNumberCyclic := _AxisReference^.Data.CallNumberCyclic + INT#2;
                        MC_MoveAdditiveCallNumber := _AxisReference^.Data.CallNumberCyclic;
                        _AxisReference^.Data.WriteCommand:= TRUE;
                        _AxisReference^.Data.HomingReq:= FALSE;
            (*			Axis.Data.DriveStopReq:= FALSE;*)
                        _AxisReference^.Data.DriveHaltReq := FALSE;
                        _AxisReference^.Data.MoveVelocityReq:= FALSE;
                        _AxisReference^.Data.TorqueControlReq:= FALSE;
                        _AxisReference^.Data.Relative:= TRUE;
                        _AxisReference^.Data.Additive:= FALSE;
                        _AxisReference^.Data.Position := Distance;
                        _AxisReference^.Data.Velocity := Velocity;
                        _AxisReference^.Data.Acceleration := Acceleration;
                        _AxisReference^.Data.Deceleration := Deceleration;
                        _AxisReference^.Data.Jerk:= Jerk;
                        MC_MoveAdditiveDone_ := FALSE;
                        MC_MoveAdditiveActive_ := TRUE;
                        MC_MoveAdditiveError_ := FALSE;
                        MC_MoveAdditiveErrorID_ :=	AXOpen.Components.Rexroth.Drives.eAxoIndraDriveErrorCode#NONE_ERROR;
                    END_IF;
                ELSE
                    MC_MoveAdditiveCallNumber := MC_MoveAdditiveCallNumber - INT#1;
                    MC_MoveAdditiveError_ := TRUE;
                    MC_MoveAdditiveErrorID_ := AXOpen.Components.Rexroth.Drives.eAxoIndraDriveErrorCode#RESOURCE_ERROR;
                END_IF;
            END_IF;
            (************** reset of outputs *************************************)
            IF Execute = FALSE THEN
                MC_MoveAdditiveCommandAborted_ := FALSE;
                MC_MoveAdditiveDone_ := FALSE;
                MC_MoveAdditiveError_ := FALSE;
                MC_MoveAdditiveErrorID_ :=	AXOpen.Components.Rexroth.Drives.eAxoIndraDriveErrorCode#NONE_ERROR;
                MC_MoveAdditiveDistance_PV := 0;
            END_IF;
            (*************** detection of command finished *******************)
            IF MC_MoveAdditiveFirstCall THEN
                IF MC_MoveAdditiveCallNumber = _AxisReference^.Data.CallNumberCyclic THEN
                    MC_MoveAdditiveActive_ := TRUE;
                    _AxisReference^.Data.CallAxis := TRUE;
                    _AxisReference^.Data.ReadOnlyData := FALSE;
                    THIS.FieldBusCommunication(AxisRef := _AxisReference,CommandWriteActive=> Dummy);
                    IF NOT _AxisReference^.Data.CommandWriteActive THEN
                        MC_MoveAdditiveActive_ := TRUE;
                        IF MC_MoveAdditiveContinuousUpdate_PV AND
                            (MC_MoveAdditiveDistance_PV<> Distance OR
                            _AxisReference^.Data.Velocity <> Velocity OR
                            _AxisReference^.Data.Acceleration <> Acceleration OR
                            _AxisReference^.Data.Deceleration <> Deceleration OR
                            _AxisReference^.Data.Jerk <> Jerk ) THEN
                            _AxisReference^.Data.Position := Distance-MC_MoveAdditiveDistance_PV;
                            _AxisReference^.Data.Velocity := Velocity;
                            _AxisReference^.Data.Acceleration := Acceleration;
                            _AxisReference^.Data.Deceleration := Deceleration;
                            _AxisReference^.Data.Jerk:= Jerk;
                            _AxisReference^.Data.WriteCommand := TRUE;
                            _AxisReference^.Data.CallAxis := TRUE;
                            _AxisReference^.Data.ReadOnlyData := FALSE;
                            MC_MoveAdditiveDistance_PV := Distance;
                            THIS.FieldBusCommunication(AxisRef := _AxisReference,CommandWriteActive=> Dummy);
                            RETURN;
                        END_IF;

                        IF _AxisReference^.Data.SetpointReached THEN
                            MC_MoveAdditiveDone_ := TRUE;
                            MC_MoveAdditiveActive_ := FALSE;
                            MC_MoveAdditiveCallNumber := MC_MoveAdditiveCallNumber - INT#1; (*Reset MC_MoveAdditiveCallNumber because reset Done *)
                        END_IF;
                    END_IF;
                    IF _AxisReference^.Data.Error THEN
                        MC_MoveAdditiveCallNumber := MC_MoveAdditiveCallNumber - INT#1;
                        MC_MoveAdditiveActive_ := FALSE;
                        MC_MoveAdditiveError_ := TRUE;
                        MC_MoveAdditiveErrorID_ := _AxisReference^.Data.ErrorID;
                    ELSIF _AxisReference^.Data.CallAxis THEN
                        MC_MoveAdditiveCallNumber := MC_MoveAdditiveCallNumber - INT#1;
                        MC_MoveAdditiveActive_ := FALSE;
                        MC_MoveAdditiveError_ := TRUE;
                        MC_MoveAdditiveErrorID_ := AXOpen.Components.Rexroth.Drives.eAxoIndraDriveErrorCode#RESOURCE_ERROR;
                    END_IF;
                ELSE
                    (*************** detection of command aborted ********************)
                    IF MC_MoveAdditiveActive_ THEN
                        MC_MoveAdditiveCommandAborted_ := TRUE;
                    END_IF;
                    MC_MoveAdditiveActive_ := FALSE;
                END_IF;
            END_IF;

            IF NOT ContinuousUpdate THEN
                MC_MoveAdditiveContinuousUpdate_PV := FALSE;
            END_IF;
            MC_MoveAdditiveExecute_PV := Execute;

            Done			:=	MC_MoveAdditiveDone_;
            Busy			:=	Execute AND NOT Done AND NOT Error;
            Active			:=	MC_MoveAdditiveActive_;
            CommandAborted	:=	MC_MoveAdditiveCommandAborted_;
            Error			:=	MC_MoveAdditiveError_;
            ErrorID			:=	TO_DINT(MC_MoveAdditiveErrorID_);
        END_METHOD

        ///<summary>
        /// This method commands a never ending controlled motion at a specified velocity.
        ///<summary>
        VAR INTERNAL
            MC_MoveVelocityExecute_PV			: 	BOOL := FALSE;		//Execute - previous value
            MC_MoveVelocityCallNumber			: 	INT; 				//Call number of the method MC_MoveVelocity
            MC_MoveVelocityFirstCall			: 	BOOL;				//First call of the method MC_MoveVelocity
            MC_MoveVelocityActive_				:	BOOL;
            MC_MoveVelocityCommandAborted_		:	BOOL;
            MC_MoveVelocityError_				:   BOOL;
            MC_MoveVelocityErrorID_				:   eAxoIndraDriveErrorCode;
            MC_MoveVelocityContinuousUpdate_PV	:   BOOL;
        END_VAR
        METHOD PUBLIC OVERRIDE MC_MoveVelocity
            VAR_INPUT
                AxisRef         :   AXOpen.Components.Abstractions.Drives.IAxoAxisReference;
                Execute         :   BOOL;                       //  Start the motion at rising edge
                ContinuousUpdate:   BOOL;                       //  Activate ‘ContinuousUpdate’ - target parameters should be changed during movement
                Velocity        :   LREAL;                      //  Value of the maximum velocity [u/s]. Can be a signed value.
                Acceleration    :   LREAL;                      //  Value of the ‘Acceleration’ (always positive) (increasing energy of the motor) [u/s2]
                Deceleration    :   LREAL;                      //  Value of the ‘Deceleration’ (always positive) (decreasing energy of the motor) [u/s2]
                Jerk            :   LREAL;                      //  Value of the ‘Jerk’ [u/s3]
                Direction       :   AXOpen.Components.Abstractions.Drives.eAxoDriveDirection;         //  Enum type (1-of-3 values: PositiveDirection, NegativeDirection, and CurrentDirection. Note: shortest way not applicable)
            END_VAR
            VAR_OUTPUT
                InVelocity      :   BOOL;                       // Commanded velocity reached
                Busy            :   BOOL;                       // The method is not finished and new output values are to be expected
                Active          :   BOOL;                       // Indicates that the method has control on the axis
                CommandAborted  :   BOOL;                       // ‘Command’ is aborted by another command
                Error           :   BOOL;                       // Signals that an error has occurred within the method
                ErrorID         :   DINT;                       // Error identification
            END_VAR
            VAR
                _AxisReference :  REF_TO AXOpen.Components.Rexroth.Drives.AxoIndraDriveAxisReference;
                Dummy : BOOL;
                Velocity_        :   LREAL;
            END_VAR

            _AxisReference ?= AxisRef;

            Messenger.ActivateOnCondition(ULINT#1408,_AxisReference = NULL, eAxoMessageCategory#ProgrammingError);

            IF(_AxisReference = NULL) THEN
                RETURN;
            END_IF;

            Messenger.ActivateOnCondition(ULINT#1429,Direction <> AXOpen.Components.Abstractions.Drives.eAxoDriveDirection#PositiveDirection AND Direction <> AXOpen.Components.Abstractions.Drives.eAxoDriveDirection#NegativeDirection, eAxoMessageCategory#ProgrammingError);

            IF Direction = AXOpen.Components.Abstractions.Drives.eAxoDriveDirection#PositiveDirection THEN
                Velocity_ := Velocity;
            ELSIF Direction = AXOpen.Components.Abstractions.Drives.eAxoDriveDirection#NegativeDirection THEN
                Velocity_ := -1 * Velocity;
            ELSE
                RETURN;
            END_IF;

            IF Execute OR (NOT Execute AND MC_MoveVelocityExecute_PV) THEN (*detection of falling edge execute*)
                MC_MoveVelocityFirstCall := TRUE;
                IF _AxisReference^.Data.CheckAccessOK THEN
                    IF Execute AND NOT MC_MoveVelocityExecute_PV THEN (*	raising edge of EXECUTE *)
                        MC_MoveVelocityContinuousUpdate_PV := ContinuousUpdate;
                        _AxisReference^.Data.CallNumberCyclic := _AxisReference^.Data.CallNumberCyclic + INT#2;
                        MC_MoveVelocityCallNumber := _AxisReference^.Data.CallNumberCyclic;
                        _AxisReference^.Data.WriteCommand:= TRUE;
                        _AxisReference^.Data.HomingReq:= FALSE;
            (*			Axis.Data.DriveStopReq:= FALSE;*)
                        _AxisReference^.Data.DriveHaltReq := FALSE;
                        _AxisReference^.Data.MoveVelocityReq:= TRUE;
                        _AxisReference^.Data.TorqueControlReq:= FALSE;
                        _AxisReference^.Data.Relative:= FALSE;
                        _AxisReference^.Data.Additive:= FALSE;
                        _AxisReference^.Data.Position:= 0;
                        _AxisReference^.Data.Velocity := Velocity_;
                        _AxisReference^.Data.Acceleration := Acceleration;
                        _AxisReference^.Data.Deceleration := Deceleration;
                        _AxisReference^.Data.Jerk:= Jerk;
                        MC_MoveVelocityActive_ := TRUE;
                        MC_MoveVelocityError_ := FALSE;
                        MC_MoveVelocityErrorID_ :=	 AXOpen.Components.Rexroth.Drives.eAxoIndraDriveErrorCode#NONE_ERROR;
                    END_IF;
                ELSE
                    MC_MoveVelocityCallNumber := MC_MoveVelocityCallNumber - INT#1;
                    MC_MoveVelocityError_ := TRUE;
                    MC_MoveVelocityErrorID_ :=  AXOpen.Components.Rexroth.Drives.eAxoIndraDriveErrorCode#RESOURCE_ERROR;
                END_IF;
            END_IF;
            (************** reset of outputs *************************************)
            IF Execute = FALSE THEN
                MC_MoveVelocityCommandAborted_ := FALSE;
                MC_MoveVelocityError_ := FALSE;
                MC_MoveVelocityErrorID_ :=	 AXOpen.Components.Rexroth.Drives.eAxoIndraDriveErrorCode#NONE_ERROR;
            END_IF;
            (*************** detection of command finished *******************)
            IF MC_MoveVelocityFirstCall THEN
                IF MC_MoveVelocityCallNumber = _AxisReference^.Data.CallNumberCyclic THEN
                    MC_MoveVelocityActive_ := TRUE;
                    _AxisReference^.Data.CallAxis := TRUE;
                    _AxisReference^.Data.ReadOnlyData := FALSE;
                    THIS.FieldBusCommunication(AxisRef := _AxisReference,CommandWriteActive=> Dummy);
                    IF NOT _AxisReference^.Data.CommandWriteActive THEN
                        MC_MoveVelocityActive_ := TRUE;
                        IF MC_MoveVelocityContinuousUpdate_PV AND
                            (_AxisReference^.Data.Velocity <> Velocity_ OR
                            _AxisReference^.Data.Acceleration <> Acceleration OR
                            _AxisReference^.Data.Deceleration <> Deceleration OR
                            _AxisReference^.Data.Jerk <> Jerk ) THEN
                            _AxisReference^.Data.Velocity := Velocity;
                            _AxisReference^.Data.Acceleration := Acceleration;
                            _AxisReference^.Data.Deceleration := Deceleration;
                            _AxisReference^.Data.Jerk:= Jerk;
                            _AxisReference^.Data.WriteCommand := TRUE;
                            _AxisReference^.Data.CallAxis := TRUE;
                            _AxisReference^.Data.ReadOnlyData := FALSE;
                            THIS.FieldBusCommunication(AxisRef := _AxisReference,CommandWriteActive=> Dummy);
                        END_IF;

                    END_IF;
                    IF _AxisReference^.Data.Error THEN
                        MC_MoveVelocityCallNumber := MC_MoveVelocityCallNumber - INT#1;
                        MC_MoveVelocityActive_ := FALSE;
                        MC_MoveVelocityError_ := TRUE;
                        MC_MoveVelocityErrorID_ := _AxisReference^.Data.ErrorID;
                    ELSIF _AxisReference^.Data.CallAxis THEN
                        MC_MoveVelocityCallNumber := MC_MoveVelocityCallNumber - INT#1;
                        MC_MoveVelocityActive_ := FALSE;
                        MC_MoveVelocityError_ := TRUE;
                        MC_MoveVelocityErrorID_ :=  AXOpen.Components.Rexroth.Drives.eAxoIndraDriveErrorCode#RESOURCE_ERROR;
                    END_IF;
                ELSE
                    (*************** detection of command aborted ********************)
                    IF MC_MoveVelocityActive_ THEN
                        MC_MoveVelocityCommandAborted_ := TRUE;
                    END_IF;
                    MC_MoveVelocityActive_ := FALSE;
                END_IF;
            END_IF;
            MC_MoveVelocityExecute_PV := Execute;

            Active			:=   MC_MoveVelocityActive_ ;
            InVelocity		:=   Active AND _AxisReference^.Data.SetpointReached;
            Busy 			:= 	 Active AND NOT InVelocity;
            CommandAborted	:=   MC_MoveVelocityCommandAborted_;
            Error			:=   MC_MoveVelocityError_;
            ErrorID			:=   TO_DINT(MC_MoveVelocityErrorID_);
        END_METHOD

        ///<summary>
        /// This method continuously exerts a torque or force of the specified magnitude. This magnitude is
        /// approached using a defined ramp (‘TorqueRamp’), and the method sets the ‘InTorque’ output if the
        /// commanded torque level is reached. This method is applicable for force and torque. When there is no external
        /// load, force is applicable. Positive torque is in the positive direction of velocity.
        ///<summary>
        VAR INTERNAL
            MC_TorqueControlExecute_PV			: 	BOOL := FALSE;		//Execute - previous value
            MC_TorqueControlCallNumber			: 	INT; 				//Call number of the method MC_TorqueControl
            MC_TorqueControlFirstCall			: 	BOOL;				//First call of the method MC_TorqueControl
            MC_TorqueControlActive_				:	BOOL;
            MC_TorqueControlCommandAborted_		:	BOOL;
            MC_TorqueControlError_				:   BOOL;
            MC_TorqueControlErrorID_			:   eAxoIndraDriveErrorCode;
            MC_TorqueControlContinuousUpdate_PV :   BOOL;
        END_VAR
        METHOD PUBLIC OVERRIDE MC_TorqueControl
            VAR_INPUT
                AxisRef         :   AXOpen.Components.Abstractions.Drives.IAxoAxisReference;
                Execute         :   BOOL;                       //  Start the motion at rising edge
                ContinuousUpdate:   BOOL;                       //  Activate ‘ContinuousUpdate’ - target parameters should be changed during movement
                Torque          :   LREAL;                      //  Value of the torque (Torque or force in technical unit [u])
                TorqueRamp      :   LREAL;                      //  The maximum time derivative of the set value of the torque or force (in technical unit per sec. [u/s])
                PositionLimit   :   LREAL;                      //  PositionLimit
                Velocity        :   LREAL;                      //  Absolute value of the maximum velocity.
                Acceleration    :   LREAL;                      //  Value of the maximum acceleration (acceleration is applicable with same sign of torque and velocity)
                Deceleration    :   LREAL;                      //  Value of the maximum deceleration (deceleration is applicable with opposite signs of torque and velocity)
                Jerk            :   LREAL;                      //  Value of the maximum jerk
                Direction       :   AXOpen.Components.Abstractions.Drives.eAxoDriveDirection;         //  Enum type (1 of 2 values: PositiveDirection, NegativeDirection or CurrentDirection). Specifies the direction of the torque. (Note: Torque input can be signed value).
            END_VAR
            VAR_OUTPUT
                InTorque        :   BOOL;                       //  Setpoint value of torque or force equals the commandedvalue
                Busy            :   BOOL;                       //  The method is not finished and new output values are to be expected
                Active          :   BOOL;                       //  Indicates that the method has control on the axis
                CommandAborted  :   BOOL;                       //  ‘Command’ is aborted by another command
                Error           :   BOOL;                       //  Signals that an error has occurred within the method
                ErrorID         :   DINT;                       //  Error identification
            END_VAR
            VAR
                _AxisReference :  REF_TO AXOpen.Components.Rexroth.Drives.AxoIndraDriveAxisReference;
                Dummy : BOOL;
                Torque_          :   LREAL;
                PositiveDirection_  : BOOL;
            END_VAR

            _AxisReference ?= AxisRef;

            Messenger.ActivateOnCondition(ULINT#1409,_AxisReference = NULL, eAxoMessageCategory#ProgrammingError);

            IF(_AxisReference = NULL) THEN
                RETURN;
            END_IF;

            Messenger.ActivateOnCondition(ULINT#1430,Direction <> AXOpen.Components.Abstractions.Drives.eAxoDriveDirection#PositiveDirection AND Direction <> AXOpen.Components.Abstractions.Drives.eAxoDriveDirection#NegativeDirection, eAxoMessageCategory#ProgrammingError);

            IF Direction = AXOpen.Components.Abstractions.Drives.eAxoDriveDirection#PositiveDirection THEN
                Torque_ := Torque;
            ELSIF Direction = AXOpen.Components.Abstractions.Drives.eAxoDriveDirection#NegativeDirection THEN
                Torque_ := -1 * Torque;
            ELSE
                RETURN;
            END_IF;

            PositiveDirection_ := Torque_ > 0;

            IF Execute OR (NOT Execute AND MC_TorqueControlExecute_PV) THEN (*detection of falling edge execute*)
                MC_TorqueControlFirstCall := TRUE;
                IF PositiveDirection_  AND THIS.ActualPosition >= PositionLimit THEN
                    _AxisReference^.Data.DriveHaltReq := TRUE;
                    _AxisReference^.Data.MoveVelocityReq:= FALSE;
                    _AxisReference^.Data.TorqueControlReq:= FALSE;
                    RETURN;
                ELSIF NOT PositiveDirection_  AND THIS.ActualPosition <= PositionLimit THEN
                    _AxisReference^.Data.DriveHaltReq := TRUE;
                    _AxisReference^.Data.MoveVelocityReq:= FALSE;
                    _AxisReference^.Data.TorqueControlReq:= FALSE;
                    RETURN;
                END_IF;
                IF _AxisReference^.Data.CheckAccessOK THEN
                    IF Execute AND NOT MC_TorqueControlExecute_PV THEN (*raising edge of EXECUTE *)
                        MC_TorqueControlContinuousUpdate_PV := ContinuousUpdate;
                        _AxisReference^.Data.CallNumberCyclic := _AxisReference^.Data.CallNumberCyclic + INT#2;
                        MC_TorqueControlCallNumber := _AxisReference^.Data.CallNumberCyclic;
                        _AxisReference^.Data.WriteCommand:= TRUE;
                        _AxisReference^.Data.HomingReq:= FALSE;
            (*			Axis.Data.DriveStopReq:= FALSE;*)
                        _AxisReference^.Data.DriveHaltReq := FALSE;
                        _AxisReference^.Data.MoveVelocityReq:= FALSE;
                        _AxisReference^.Data.TorqueControlReq:= TRUE;
                        _AxisReference^.Data.Relative:= FALSE;
                        _AxisReference^.Data.Additive:= FALSE;
                        _AxisReference^.Data.Position:= 0;
                        _AxisReference^.Data.Velocity := Velocity;
                        _AxisReference^.Data.Acceleration := Acceleration;
                        _AxisReference^.Data.Deceleration := Deceleration;
                        _AxisReference^.Data.Jerk:= Jerk;
                        _AxisReference^.Data.Torque:= Torque_;
                        MC_TorqueControlActive_ := TRUE;
                        MC_TorqueControlError_ := FALSE;
                        MC_TorqueControlErrorID_ :=	 AXOpen.Components.Rexroth.Drives.eAxoIndraDriveErrorCode#NONE_ERROR;
                    END_IF;
                ELSE
                    MC_TorqueControlCallNumber := MC_TorqueControlCallNumber - INT#1;
                    MC_TorqueControlError_ := TRUE;
                    MC_TorqueControlErrorID_ :=  AXOpen.Components.Rexroth.Drives.eAxoIndraDriveErrorCode#RESOURCE_ERROR;
                END_IF;
            END_IF;
            (************** reset of outputs *************************************)
            IF Execute = FALSE THEN
                MC_TorqueControlCommandAborted_ := FALSE;
                MC_TorqueControlError_ := FALSE;
                MC_TorqueControlErrorID_ :=	 AXOpen.Components.Rexroth.Drives.eAxoIndraDriveErrorCode#NONE_ERROR;
            END_IF;
            (*************** detection of command finished *******************)
            IF MC_TorqueControlFirstCall THEN
                IF MC_TorqueControlCallNumber = _AxisReference^.Data.CallNumberCyclic THEN
                    MC_TorqueControlActive_ := TRUE;
                    _AxisReference^.Data.CallAxis := TRUE;
                    _AxisReference^.Data.ReadOnlyData := FALSE;
                    THIS.FieldBusCommunication(AxisRef := _AxisReference,CommandWriteActive=> Dummy);
                    IF NOT _AxisReference^.Data.CommandWriteActive THEN
                        MC_TorqueControlActive_ := TRUE;
                        IF MC_TorqueControlContinuousUpdate_PV AND
                            (_AxisReference^.Data.Torque <> Torque_ OR
                            // _AxisReference^.Data.TorqueRamp <> TorqueRamp OR
                            _AxisReference^.Data.Velocity <> Velocity OR
                            _AxisReference^.Data.Acceleration <> Acceleration OR
                            _AxisReference^.Data.Deceleration <> Deceleration OR
                            _AxisReference^.Data.Jerk <> Jerk ) THEN
                            _AxisReference^.Data.Torque := Torque_ ;
                            _AxisReference^.Data.Velocity := Velocity;
                            _AxisReference^.Data.Acceleration := Acceleration;
                            _AxisReference^.Data.Deceleration := Deceleration;
                            _AxisReference^.Data.Jerk:= Jerk;
                            _AxisReference^.Data.WriteCommand := TRUE;
                            _AxisReference^.Data.CallAxis := TRUE;
                            _AxisReference^.Data.ReadOnlyData := FALSE;
                            THIS.FieldBusCommunication(AxisRef := _AxisReference,CommandWriteActive=> Dummy);
                        END_IF;

                    END_IF;
                    IF _AxisReference^.Data.Error THEN
                        MC_TorqueControlCallNumber := MC_TorqueControlCallNumber - INT#1;
                        MC_TorqueControlActive_ := FALSE;
                        MC_TorqueControlError_ := TRUE;
                        MC_TorqueControlErrorID_ := _AxisReference^.Data.ErrorID;
                    ELSIF _AxisReference^.Data.CallAxis THEN
                        MC_TorqueControlCallNumber := MC_TorqueControlCallNumber - INT#1;
                        MC_TorqueControlActive_ := FALSE;
                        MC_TorqueControlError_ := TRUE;
                        MC_TorqueControlErrorID_ :=  AXOpen.Components.Rexroth.Drives.eAxoIndraDriveErrorCode#RESOURCE_ERROR;
                    END_IF;
                ELSE
                    (*************** detection of command aborted ********************)
                    IF MC_TorqueControlActive_ THEN
                        MC_TorqueControlCommandAborted_ := TRUE;
                    END_IF;
                    MC_TorqueControlActive_ := FALSE;
                END_IF;
            END_IF;
            MC_TorqueControlExecute_PV := Execute;

            Active			:=   MC_TorqueControlActive_;
            InTorque		:=   Active AND _AxisReference^.Data.SetpointReached;
            Busy 			:= 	 Active AND NOT InTorque;
            CommandAborted	:=   MC_TorqueControlCommandAborted_;
            Error			:=   MC_TorqueControlError_;
            ErrorID			:=   TO_DINT(MC_TorqueControlErrorID_);

        END_METHOD

        ///<summary>
        /// This method shifts the coordinate system of an axis by manipulating both the set-point position as well as the
        /// actual position of an axis with the same value without any movement caused. (Re-calibration with same following error).
        /// This can be used for instance for a reference situation. This method can also be used during motion without changing
        /// the commanded position, which is now positioned in the shifted coordinate system.
        ///<summary>
        VAR INTERNAL
            MC_SetPositionDone_					:	BOOL;
            MC_SetPositionBusy_					:	BOOL;
            MC_SetPositionError_ 				:	BOOL;
            MC_SetPositionErrorID_ 				:	eAxoIndraDriveErrorCode;
            MC_SetPositionState_ 				:	UINT;
            MC_SetPositionValue_ 				:	DINT;
        END_VAR
        METHOD PUBLIC OVERRIDE MC_SetPosition
            VAR_INPUT
                AxisRef         :   AXOpen.Components.Abstractions.Drives.IAxoAxisReference;
                Execute         :   BOOL;                       //  Start setting position in axis
                Position        :   LREAL;                       //  Position unit [u] (Means ‘Distance’ if ‘Relative’= TRUE)
                Relative        :   BOOL;                       //  ‘Relative’ distance if True, ‘Absolute’ position if False (= Default)
                ExecutionMode   :   AXOpen.Components.Abstractions.Drives.eAxoExecutionMode;          //  Defines the chronological sequence of the method.
            END_VAR
            VAR_OUTPUT
                Done            :   BOOL;                       //  ‘Position’ has new value
                Busy            :   BOOL;                       //  The method is not finished and new output values are to be expected
                Error           :   BOOL;                       //  Signals that an error has occurred within the method
                ErrorID         :   DINT;                       //  Error identification
            END_VAR
            VAR
                _AxisReference :  REF_TO AXOpen.Components.Rexroth.Drives.AxoIndraDriveAxisReference;
                Dummy : BOOL;
                _result : AXOpen.Core.IAxoTaskState;
                _ErrorID    :   eAxoIndraDriveErrorCode;
                _Valid  :   BOOL;
                _Error  :   BOOL;
                _Position   :   LREAL;
                _dint       :   DINT;
            END_VAR

            _AxisReference ?= AxisRef;

            Messenger.ActivateOnCondition(ULINT#1410 ,_AxisReference = NULL, eAxoMessageCategory#ProgrammingError);

            IF(_AxisReference = NULL) THEN
                RETURN;
            END_IF;

            IF Execute THEN
                IF MC_SetPositionState_ = UINT#0 THEN
                    MC_SetPositionDone_ := FALSE;
                    MC_SetPositionBusy_ := TRUE;
                    MC_SetPositionError_ := FALSE;
                    MC_SetPositionErrorID_ := AXOpen.Components.Rexroth.Drives.eAxoIndraDriveErrorCode#NONE_ERROR;
                    MC_SetPositionValue_ := 0;
                    MC_SetPositionState_ := MC_SetPositionState_ + UINT#10;
                END_IF;
            END_IF;
            IF MC_SetPositionState_ = UINT#10 THEN
                IF ExecutionMode = AXOpen.Components.Abstractions.Drives.eAxoExecutionMode#Immediately OR ExecutionMode =AXOpen.Components.Abstractions.Drives.eAxoExecutionMode#Queued AND _AxisReference^.Data.Standstill THEN
                    IF Relative THEN
                        MC_SetPositionValue_ := MC_SetPositionValue_ + TO_DINT(Position * EXP(LN(10)*PositionExponent));
                        MC_SetPositionState_ := MC_SetPositionState_ + UINT#30;
                    ELSE
                        MC_SetPositionValue_ := MC_SetPositionValue_ + TO_DINT(Position * EXP(LN(10)*PositionExponent));
                        MC_SetPositionState_ := MC_SetPositionState_ + UINT#10;
                    END_IF;
                END_IF;
            END_IF;
            IF MC_SetPositionState_ = UINT#20 THEN
                THIS.AxoReadActualPosition(Enable := TRUE,Valid => _Valid, Error => _Error, ErrorID => _dint, Position => _Position);
                _ErrorID := TO_WORD(_dint);
                IF _Error THEN
                    MC_SetPositionError_ 		:= TRUE;
                    MC_SetPositionErrorID_ 		:= _ErrorID;
                END_IF;
                IF _Valid THEN
                    MC_SetPositionValue_ := MC_SetPositionValue_ - TO_DINT((_Position ) * EXP(LN(10)*PositionExponent));
                    MC_SetPositionState_ := MC_SetPositionState_ + UINT#10;
                END_IF;
            END_IF;
            IF MC_SetPositionState_ = UINT#30 THEN
                THIS.AxoReadActualPosition(Enable := FALSE,Valid => _Valid, Error => _Error,ErrorID => _dint, Position => _Position);
                _ErrorID := TO_WORD(_dint);
                IF NOT _Valid THEN
                    MC_SetPositionState_ := MC_SetPositionState_ + UINT#10;
                END_IF;
            END_IF;
            IF MC_SetPositionState_ = UINT#40 THEN
                //S-0-0275, Coordinate offset value
                _result := THIS.AxoWriteParameter(ParameterNumber := 275, Value := MC_SetPositionValue_ ,ExecutionMode := AXOpen.Components.Abstractions.Drives.eAxoExecutionMode#Immediately, ErrorID =>_dint);
                _ErrorID := TO_WORD(_dint);
                IF _result.IsDone() THEN
                    MC_SetPositionState_ := MC_SetPositionState_ + UINT#10;
                END_IF;
                IF _result.HasError() THEN
                    MC_SetPositionError_ 		:= TRUE;
                    MC_SetPositionErrorID_ 		:= _ErrorID;
                END_IF;
            END_IF;
            IF MC_SetPositionState_ = UINT#50 THEN
                AxoWriteParameter_Task.Restore();
                IF(AxoWriteParameter_Task.IsReady()) THEN
                    MC_SetPositionState_ := MC_SetPositionState_ + UINT#10;
                    RETURN;
                END_IF;
            END_IF;
            IF MC_SetPositionState_ = UINT#60 THEN
                //S-0-0199, C3400 Shift coordinate system procedure command
                _result := THIS.AxoWriteParameter(ParameterNumber := 199, Value := 3 ,ExecutionMode := AXOpen.Components.Abstractions.Drives.eAxoExecutionMode#Immediately, ErrorID =>_dint);
                _ErrorID := TO_WORD(_dint);
                IF _result.IsDone() THEN
                    MC_SetPositionState_ := MC_SetPositionState_ + UINT#10;
                END_IF;
                IF _result.HasError() THEN
                    MC_SetPositionError_ 		:= TRUE;
                    MC_SetPositionErrorID_ 		:= _ErrorID;
                END_IF;
            END_IF;
            IF MC_SetPositionState_ = UINT#70 THEN
                AxoWriteParameter_Task.Restore();
                IF(AxoWriteParameter_Task.IsReady()) THEN
                    MC_SetPositionState_ := MC_SetPositionState_ + UINT#10;
                    RETURN;
                END_IF;
            END_IF;
            IF MC_SetPositionState_ = UINT#80 THEN
                //S-0-0199, C3400 Shift coordinate system procedure command
                _result := THIS.AxoWriteParameter(ParameterNumber := 199, Value := 0 ,ExecutionMode := AXOpen.Components.Abstractions.Drives.eAxoExecutionMode#Immediately, ErrorID =>_dint);
                _ErrorID := TO_WORD(_dint);
                IF _result.IsDone() THEN
                    MC_SetPositionState_ := MC_SetPositionState_ + UINT#10;
                END_IF;
                IF _result.HasError() THEN
                    MC_SetPositionError_ 		:= TRUE;
                    MC_SetPositionErrorID_ 		:= _ErrorID;
                END_IF;
            END_IF;
            IF MC_SetPositionState_ = UINT#90 THEN
                AxoWriteParameter_Task.Restore();
                IF(AxoWriteParameter_Task.IsReady()) THEN
                    MC_SetPositionState_ := MC_SetPositionState_ + UINT#10;
                    RETURN;
                END_IF;
            END_IF;

            IF MC_SetPositionState_ = UINT#100 THEN
                MC_SetPositionDone_ := TRUE;
                MC_SetPositionBusy_ := FALSE;
            END_IF;

            Done				:=	MC_SetPositionDone_;
            Busy 				:=	MC_SetPositionBusy_;
            Error 				:=	MC_SetPositionError_;
            ErrorID 			:=	TO_DINT(MC_SetPositionErrorID_);

            IF NOT Execute THEN
                MC_SetPositionDone_ := FALSE;
                MC_SetPositionBusy_ := FALSE;
                MC_SetPositionError_ := FALSE;
                MC_SetPositionErrorID_ := AXOpen.Components.Rexroth.Drives.eAxoIndraDriveErrorCode#NONE_ERROR;
                MC_SetPositionState_ := UINT#0;
            END_IF;
        END_METHOD

        ///<summary>
        /// This method sets the values of override for the whole axis, and all functions that are working on that axis. The override
        /// parameters contribute as a factor to the calculation of the commanded velocity, acceleration and jerk of the motion.
        ///<summary>
        METHOD PUBLIC OVERRIDE MC_SetOverride
            VAR_INPUT
                AxisRef         :   AXOpen.Components.Abstractions.Drives.IAxoAxisReference;
                Enable          :   BOOL;                       //  If SET, it writes the value of the override factor continuously. If RESET it should keep the last value.
                VelocityFactor  :   LREAL;                      //  New override factor for the velocity
                AccelerationFactor:   LREAL;                    //  New override factor for the acceleration/deceleration
                JerkFactor      :   LREAL;                      //  New override factor for the jer
            END_VAR
            VAR_OUTPUT
                Enabled         :   BOOL;                       //  Signals that the override factor(s) is (are) set successfully
                Busy            :   BOOL;                       //  The method is not finished and new output values are to be expected
                Error           :   BOOL;                       //  Signals that an error has occurred within the method
                ErrorID         :   DINT;                       //  Error identification
            END_VAR
            VAR
                _AxisReference :  REF_TO AXOpen.Components.Rexroth.Drives.AxoIndraDriveAxisReference;
                Dummy : BOOL;
            END_VAR

            _AxisReference ?= AxisRef;

            Messenger.ActivateOnCondition(ULINT#1411,_AxisReference = NULL, eAxoMessageCategory#ProgrammingError);

            IF(_AxisReference = NULL) THEN
                RETURN;
            END_IF;

            IF Enable THEN
                Busy := TRUE;
                IF _AxisReference^.Data.CheckAccessOK	THEN
                    IF VelocityFactor <= 0.0 OR  VelocityFactor > 1.0 OR AccelerationFactor <= 0.0 OR  AccelerationFactor > 1.0 OR JerkFactor <= 0.0 OR  JerkFactor > 1.0 THEN
                        Enabled	:= FALSE;
                        Busy := FALSE;
                        Error := TRUE;
                        ErrorID:= TO_DINT(AXOpen.Components.Rexroth.Drives.eAxoIndraDriveErrorCode#INPUT_RANGE_ERROR);
                    ELSE
                        _AxisReference^.Data.CallAxis := TRUE;
                        IF _AxisReference^.Data.OverrideVelocityFactor <> VelocityFactor OR _AxisReference^.Data.OverrideAccelerationFactor <> AccelerationFactor OR  _AxisReference^.Data.OverrideJerkFactor <> JerkFactor THEN
                            _AxisReference^.Data.OverrideVelocityFactor := VelocityFactor;
                            _AxisReference^.Data.OverrideAccelerationFactor := AccelerationFactor;
                            _AxisReference^.Data.OverrideJerkFactor := JerkFactor;
                            _AxisReference^.Data.WriteCommand := TRUE;
                        END_IF;;
                        _AxisReference^.Data.ReadOnlyData := FALSE;
                        THIS.FieldBusCommunication(AxisRef := _AxisReference, CommandWriteActive=> Dummy);
                        Enabled := TRUE;
                        Busy := FALSE;
                        Error := FALSE;
                        ErrorID := TO_DINT(AXOpen.Components.Rexroth.Drives.eAxoIndraDriveErrorCode#NONE_ERROR);
                    END_IF;
                ELSE
                    Enabled	:= FALSE;
                    Busy := FALSE;
                    Error := TRUE;
                    ErrorID := TO_DINT(AXOpen.Components.Rexroth.Drives.eAxoIndraDriveErrorCode#RESOURCE_ERROR);
                END_IF;
            ELSE
                Enabled	:= FALSE;
                Busy := FALSE;
                Error := FALSE;
                ErrorID := TO_DINT(AXOpen.Components.Rexroth.Drives.eAxoIndraDriveErrorCode#NONE_ERROR);
            END_IF;

        END_METHOD

        ///<summary>
        /// This method returns the value of a vendor specific parameter. The returned Value has to be converted to Real
        /// if necessary. If not possible, the vendor has to supply a vendor specific method to read the parameter.
        ///<summary>
        VAR INTERNAL
            MC_ReadParameterEnable_PV			: 	BOOL := FALSE;		//Enable - previous value
            MC_ReadParameterDone_PV				:	BOOL := FALSE;		//Done - previous value
            MC_ReadParameterCallNumber			: 	INT; 				//Call number of the method MC_ReadParameter
            MC_ReadParameterNumber_PV			: 	DINT;				//ParameterNumber - previous value (stored at rising edge of the Enable)
            MC_ReadParameterFirstCall			: 	BOOL;				//First call of the method MC_ReadParameter
            MC_ReadParameterDone_				:	BOOL;
            MC_ReadParameterActive_				:	BOOL := FALSE;
            MC_ReadParameterError_				:	BOOL;
            MC_ReadParameterErrorID_			:	eAxoIndraDriveErrorCode;
            MC_ReadParameterValue_				:	DINT;
        END_VAR
        METHOD PUBLIC OVERRIDE MC_ReadParameter
            VAR_INPUT
                AxisRef         :   AXOpen.Components.Abstractions.Drives.IAxoAxisReference;
                Enable          :   BOOL;                       //  Get the value of the parameter continuously while enabled
                ParameterNumber :   DINT;                       //  Number of the parameter. One can also use symbolic parameter names which are declared as VAR CONST.
            END_VAR
            VAR_OUTPUT
                Valid           :   BOOL;                       //  A valid output is available at the method
                Busy            :   BOOL;                       //  The method is not finished and new output values are to be expected
                Error           :   BOOL;                       //  Signals that an error has occurred within the method
                ErrorID         :   DINT;                       //  Error identification
                Value           :   LINT;                       //  Value of the specified parameter in the datatype, as specified by the vendor
            END_VAR
            VAR
                _AxisReference :  REF_TO AXOpen.Components.Rexroth.Drives.AxoIndraDriveAxisReference;
                Dummy : BOOL;
            END_VAR

            _AxisReference ?= AxisRef;

            Messenger.ActivateOnCondition(ULINT#1412,_AxisReference = NULL, eAxoMessageCategory#ProgrammingError);

            IF(_AxisReference = NULL) THEN
                RETURN;
            END_IF;

            IF Enable THEN
                MC_ReadParameterFirstCall := TRUE;
                IF _AxisReference^.Data.CheckAccessOK THEN
                    IF Enable AND NOT MC_ReadParameterEnable_PV THEN(*	raising edge of Enable *)
                        IF NOT _AxisReference^.Data.ActiveAcyclicCommunication THEN
                            _AxisReference^.Data.CallNumberAcyclic := _AxisReference^.Data.CallNumberAcyclic + INT#2;
                            MC_ReadParameterCallNumber := _AxisReference^.Data.CallNumberAcyclic;
                            MC_ReadParameterNumber_PV := ParameterNumber;
                            _AxisReference^.Data.WriteParameter := FALSE;
                            _AxisReference^.Data.SelectDataType := UINT#1;
                            _AxisReference^.Data.ParameterNumber := MC_ReadParameterNumber_PV;
                            MC_ReadParameterError_ := FALSE;
                            MC_ReadParameterErrorID_ := AXOpen.Components.Rexroth.Drives.eAxoIndraDriveErrorCode#NONE_ERROR;
                        ELSE
                            MC_ReadParameterError_ := TRUE;
                            MC_ReadParameterErrorID_ := AXOpen.Components.Rexroth.Drives.eAxoIndraDriveErrorCode#ACCESS_ERROR;
                        END_IF;
                    END_IF;
                ELSE
                    MC_ReadParameterCallNumber := MC_ReadParameterCallNumber - INT#1;
                    MC_ReadParameterError_ := TRUE;
                    MC_ReadParameterErrorID_ := AXOpen.Components.Rexroth.Drives.eAxoIndraDriveErrorCode#RESOURCE_ERROR;
                END_IF;
            END_IF;
            IF MC_ReadParameterFirstCall THEN
                IF MC_ReadParameterCallNumber = _AxisReference^.Data.CallNumberAcyclic AND Enable	THEN
                    _AxisReference^.Data.CallAxisParameterMethod := TRUE;
                    _AxisReference^.Data.EnableAcyclicCommunication := TRUE;
                    THIS.AcyclicCommunicationCall(AxisRef :=  _AxisReference , DPV1ParameterNumber := TRUE, Active => Dummy);
                    Busy := _AxisReference^.Data.ActiveAcyclicCommunication;
                    IF _AxisReference^.Data.DoneAcyclicCommunication THEN
                        MC_ReadParameterDone_ := TRUE;
                        MC_ReadParameterActive_ := FALSE;
                        MC_ReadParameterValue_ := _AxisReference^.Data.ReadValueDint;
                    END_IF;
                    IF _AxisReference^.Data.Error_AcyclicCommunication THEN
                        MC_ReadParameterCallNumber := MC_ReadParameterCallNumber - INT#1;
                        MC_ReadParameterDone_ := FALSE;
                        MC_ReadParameterActive_ := FALSE;
                        MC_ReadParameterError_ := _AxisReference^.Data.Error_AcyclicCommunication;
                        MC_ReadParameterErrorID_ := _AxisReference^.Data.ErrorID_AcyclicCommunication;
                        _AxisReference^.Data.CallAxisParameterMethod := TRUE;
                        _AxisReference^.Data.EnableAcyclicCommunication := FALSE;
                        THIS.AcyclicCommunicationCall(AxisRef :=  _AxisReference , DPV1ParameterNumber := TRUE, Active => Dummy);
                    ELSIF  _AxisReference^.Data.CallAxisParameterMethod THEN
                        MC_ReadParameterCallNumber := MC_ReadParameterCallNumber - INT#1;
                        MC_ReadParameterDone_ := FALSE;
                        MC_ReadParameterActive_ := FALSE;
                        MC_ReadParameterError_ := TRUE;
                        MC_ReadParameterErrorID_ := AXOpen.Components.Rexroth.Drives.eAxoIndraDriveErrorCode#RESOURCE_ERROR;
                        _AxisReference^.Data.EnableAcyclicCommunication := FALSE;
                    END_IF;
                ELSIF Enable AND MC_ReadParameterEnable_PV AND MC_ReadParameterCallNumber = _AxisReference^.Data.CallNumberAcyclic THEN
                    _AxisReference^.Data.CallAxisParameterMethod := TRUE;
                    _AxisReference^.Data.EnableAcyclicCommunication := FALSE;
                    THIS.AcyclicCommunicationCall(AxisRef :=  _AxisReference , DPV1ParameterNumber := TRUE, Active => Dummy);
                    MC_ReadParameterDone_ := FALSE;
                    MC_ReadParameterActive_ := FALSE;
                    MC_ReadParameterValue_ := DINT#0;
                    MC_ReadParameterError_ := FALSE;
                    MC_ReadParameterErrorID_ := AXOpen.Components.Rexroth.Drives.eAxoIndraDriveErrorCode#NONE_ERROR;
                ELSIF NOT Enable AND MC_ReadParameterEnable_PV THEN
                    MC_ReadParameterDone_ := FALSE;
                    MC_ReadParameterActive_ := FALSE;
                    MC_ReadParameterValue_ := DINT#0;
                    MC_ReadParameterError_ := FALSE;
                    MC_ReadParameterErrorID_ := AXOpen.Components.Rexroth.Drives.eAxoIndraDriveErrorCode#NONE_ERROR;
                    _AxisReference^.Data.ActiveAcyclicCommunication := FALSE;
                    _AxisReference^.Data.DoneAcyclicCommunication := FALSE;
                END_IF;
            END_IF;
            MC_ReadParameterEnable_PV := Enable;
